FUNCTION_BLOCK AirPiston EXTENDS FBA_Drive IMPLEMENTS I_ContinuousDrive
VAR_OUTPUT
	valveExtend AT %Q* : BOOL;
	valveRetract AT %Q* : BOOL;
END_VAR
VAR //constructor
	useBrake : BOOL; //optional - set to FALSE if retraction brake pulse is not required
END_VAR
VAR
	mode : (HOLD, IN, OUT, BRAKE);
	brakePulse : TP; //generates the retraction pulse
END_VAR
VAR_STAT CONSTANT
	brakeWidth : TIME := T#650MS;
END_VAR

IF NOT bEnable THEN
	stop();
	RETURN;
END_IF

brakePulse(IN:= , PT:= brakeWidth, Q=> , ET=> ); //reversal to act as brake
brakePulse.IN := brakePulse.IN AND brakePulse.Q; //automatically turn off pulse

override(); //alters the mode to prevent exceeding limits

CASE mode OF
	HOLD:
		valveExtend := FALSE;
		valveRetract := FALSE;
		
	IN:
		valveExtend := TRUE;
		valveRetract := FALSE;
		
	OUT:
		valveExtend := FALSE;
		valveRetract := TRUE;
		
	BRAKE: //coasts past inner limit, then slides back
		valveExtend := FALSE;
		valveRetract := TRUE;
		
		IF AtInnerLimit THEN
			mode := HOLD;
		END_IF
		
END_CASE

valveRetract := valveRetract OR brakePulse.Q; //from mode or brake

PROPERTY Active : BOOL
GET
Active :=
	mode <> HOLD AND
	valveExtend OR valveRetract;
END_GET
END_PROPERTY

PROPERTY Error : BOOL
GET
END_GET
END_PROPERTY

METHOD extend : BOOL
VAR_INPUT
END_VAR
IF mode <> BRAKE THEN
	mode := IN;
END_IF
END_METHOD

METHOD homingSequence : BOOL
CASE step OF
	Homing.IDLE:
		step := Homing.START;
		
	Homing.START:
		IF AtHome THEN //if reached home
			step := Homing.DONE;
		ELSE
			mode := OUT;
		END_IF
		
	Homing.DONE:
		mode := HOLD;
		homingComplete := TRUE;
		homingSequence := TRUE;		
	
END_CASE
END_METHOD

{attribute 'TcRpcEnable'}
METHOD moveContinuous : BOOL
VAR_INPUT
	direction : MC_Direction;
END_VAR
IF direction = MC_Positive_Direction THEN
	retract();
ELSIF direction = MC_Negative_Direction THEN
	extend();
END_IF
END_METHOD

METHOD PRIVATE override : BOOL
VAR_INPUT
END_VAR
IF brakePulse.Q THEN
	mode := HOLD;
END_IF

IF AtHome AND (valveRetract OR mode = OUT) THEN
	mode := HOLD;
	
ELSIF AtInnerLimit AND (valveExtend OR mode = IN) THEN	
	brakePulse.IN := useBrake;
	mode := HOLD;
END_IF


IF NOT bEnable THEN
	stop();
END_IF
END_METHOD

METHOD reset : BOOL
VAR_INPUT
END_VAR
stop();
END_METHOD

METHOD retract : BOOL
VAR_INPUT
END_VAR
IF mode <> BRAKE THEN
	mode := OUT;
END_IF
END_METHOD

METHOD stop : BOOL
VAR_INPUT
END_VAR
valveExtend := FALSE;
valveRetract := FALSE;
mode := HOLD;
END_METHOD

METHOD toHome : BOOL
VAR_INPUT
END_VAR
mode := OUT;
END_METHOD

END_FUNCTION_BLOCK

(* stored: Version 1.1.0.1, ProductVersion 3.1.4024.11
   POU AirPiston: Id {ef8d0471-4ac2-4d12-9e08-c4e8a3719cb6}, SpecialFunc None
   Folder Properties: Id {669624c0-4281-4400-bae4-85e7fdf7ac6d}
   Property Active: Id {22957210-b761-4111-803e-aaadd405ae90}
   Get Get: Id {5b6c8e85-c34d-419a-b0de-f334097cf117}
   Property Error: Id {230cce02-1702-429c-9486-e59a94594ced}
   Get Get: Id {085385ed-a3e2-4a8f-934d-c13a4afa77c0}
   Method extend: Id {c905417d-ebb0-4426-b712-8b35f4512697}
   Method homingSequence: Id {c3ff30f8-ced2-4f8e-b758-e21ca109ec69}
   Method moveContinuous: Id {9a8898cf-5010-49f6-8f04-ca266b1a5de1}
   Method override: Id {4aec8fb7-f31e-4265-bc33-91f3ef3efeab}
   Method reset: Id {b003bfbd-7d0c-4dc3-8afd-761691b183a9}
   Method retract: Id {d6cfbb92-1846-4f17-b88f-dcdab10c19f1}
   Method stop: Id {c035c442-83bc-4f21-a06c-19730e7f9f48}
   Method toHome: Id {d81f04ec-b071-439a-ada5-0c0fda6b57f9} *)
